(* CODESYS project Controle de Nivel.project

Project tree, tasks and I/O mapping:
  Device : CODESYS Control Win V3, 3S - Smart Software Solutions GmbH, order no. 305021, version 3.5.11.30
    application Application
      libraries: Standard, * (System)
      task MainTask (cyclic, interval t#20ms, priority 1) calls PLC_PRG
      program PLC_PRG [LD]
      Symbols
*)

// Device/Application/PLC_PRG
PROGRAM PLC_PRG
VAR
	S1: BOOL;
	S2: BOOL;
	S3: BOOL;
	V1: BOOL;
	V2: BOOL;
	V3: BOOL;
	B1: BOOL;
	B2: BOOL;
	E1: BOOL;
	NIVEL: INT;
END_VAR
VAR // added by the converter: edge detectors and wires of the graphical bodies
    _w1, _w2, _w3, _w4 : BOOL;
END_VAR

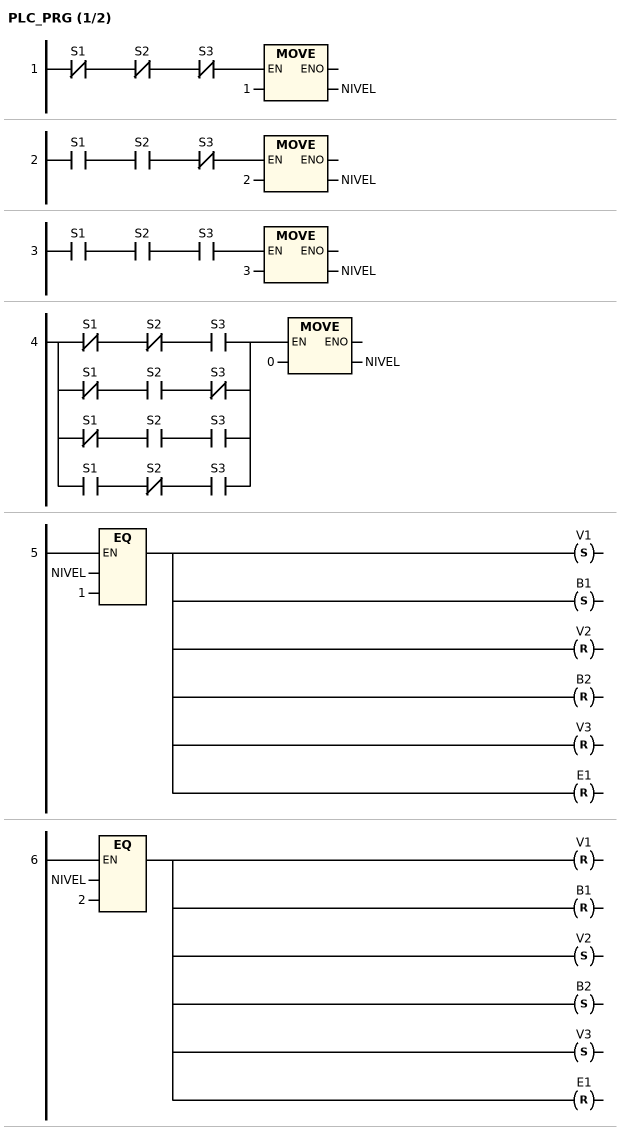
// NETWORK 1
IF NOT S1 AND NOT S2 AND NOT S3 THEN NIVEL := 1; END_IF

// NETWORK 2
IF S1 AND S2 AND NOT S3 THEN NIVEL := 2; END_IF

// NETWORK 3
IF S1 AND S2 AND S3 THEN NIVEL := 3; END_IF

// NETWORK 4
IF NOT S1 AND NOT S2 AND S3 OR NOT S1 AND S2 AND NOT S3 OR NOT S1 AND S2 AND S3 OR S1 AND NOT S2 AND S3 THEN
    NIVEL := 0;
END_IF

// NETWORK 5
_w1 := NIVEL = 1;
V1 S= _w1;
B1 S= _w1;
V2 R= _w1;
B2 R= _w1;
V3 R= _w1;
E1 R= _w1;

// NETWORK 6
_w2 := NIVEL = 2;
V1 R= _w2;
B1 R= _w2;
V2 S= _w2;
B2 S= _w2;
V3 S= _w2;
E1 R= _w2;

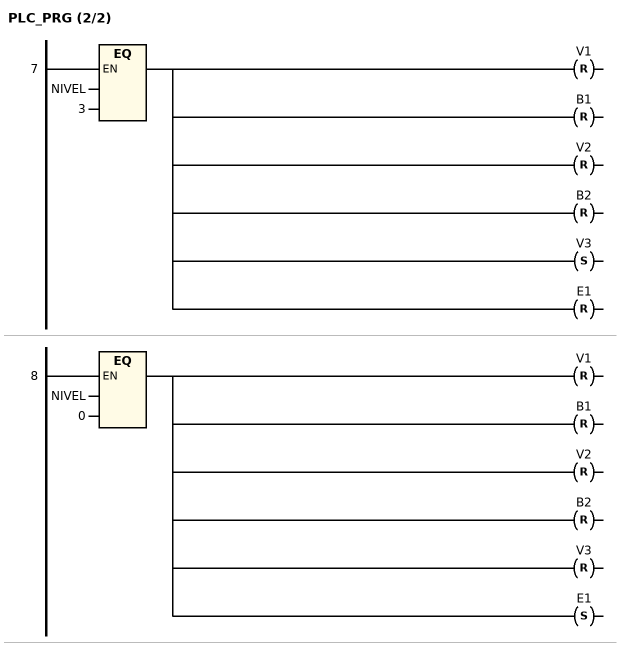
// NETWORK 7
_w3 := NIVEL = 3;
V1 R= _w3;
B1 R= _w3;
V2 R= _w3;
B2 R= _w3;
V3 S= _w3;
E1 R= _w3;

// NETWORK 8
_w4 := NIVEL = 0;
V1 R= _w4;
B1 R= _w4;
V2 R= _w4;
B2 R= _w4;
V3 R= _w4;
E1 S= _w4;

END_PROGRAM
